FUNCTION_BLOCK ABSTRACT _AbstractState EXTENDS State
VAR_INPUT
END_VAR
VAR_OUTPUT
END_VAR
VAR
	_ctx: REFERENCE TO StateContext;
END_VAR

//FB_Init is always available implicitly and it is used primarily for initialization.
//The return value is not evaluated. For a specific influence, you can also declare the
//methods explicitly and provide additional code there with the standard initialization
//code. You can evaluate the return value.
METHOD FB_Init: BOOL
VAR_INPUT
    bInitRetains: BOOL; // TRUE: the retain variables are initialized (reset warm / reset cold)
    bInCopyCode: BOOL;  // TRUE: the instance will be copied to the copy code afterward (online change)
	
	ctx: REFERENCE TO StateContext;
END_VAR
_ctx REF= ctx;
END_METHOD

END_FUNCTION_BLOCK

(* stored: Version 1.1.0.1
   POU _AbstractState: Id {8e259848-6b11-4f4c-98b7-7f0605698051}, SpecialFunc None
   Method FB_Init: Id {8de271b5-b438-4aca-a7bb-447a99209c7a} *)
